// TIA Portal V17 export
// export: Created 2024-10-17T14:16:18.5693745Z, ExportSetting WithDefaults, DisplayName Totally Integrated Automation Portal, DisplayVersion V17 Update 4, DisplayName TIA Portal Openness, DisplayVersion V17 Update 4, DisplayName TIA Portal Version Control Interface, DisplayVersion V17, DisplayName SINAMICS Startdrive Advanced, DisplayVersion V17 Update2, DisplayName SINAMICS Startdrive G130, G150, S120, S150, SINAMICS MV, S210, DisplayVersion V17 Update2, DisplayName SINAMICS Startdrive G110M, G120, G120C, G120D, G120P, G115D, DisplayVersion V17 Update2, DisplayName STEP 7 Professional, DisplayVersion V17 Update 4, DisplayName STEP 7 Safety, DisplayVersion V17, DisplayName WinCC Advanced / Unified PC, DisplayVersion V17 Update 4
TYPE "LPMLV2022_typeStatusProcessVariables"
TITLE = LPMLV2022_typeStatusProcessVariables
// Support: tech.team.motioncontrol@siemens.com
// stored: IsFailsafeCompliant false
   STRUCT
      Parameter_REAL { ExternalWritable := 'False'} : Array[0.."LPMLV2022_STATUS_PROCESS_VARIABLES_PARAMETER_REAL_UPPER_LIM"] of "LPMLV2022_typeParameter_REAL";   // Structured Array of Recipe Process Variable information for values with REAL data type
      Parameter_STRING { ExternalWritable := 'False'} : Array[0.."LPMLV2022_STATUS_PROCESS_VARIABLES_PARAMETER_STRING_UPPER_LIM"] of "LPMLV2022_typeParameter_STRING";   // Structured Array of Recipe Process Variable information for values with STRING data type
      Parameter_LREAL { ExternalWritable := 'False'} : Array[0.."LPMLV2022_STATUS_PROCESS_VARIABLES_PARAMETER_LREAL_UPPER_LIM"] of "LPMLV2022_typeParameter_LREAL";   // Structured Array of Recipe Process Variable information for values with LREAL data type
      Parameter_DINT { ExternalWritable := 'False'} : Array[0.."LPMLV2022_STATUS_PROCESS_VARIABLES_PARAMETER_DINT_UPPER_LIM"] of "LPMLV2022_typeParameter_DINT";   // Structured Array of Recipe Process Variable Information for values with DINT data type
      Parameter_BOOL { ExternalWritable := 'False'} : Array[0.."LPMLV2022_STATUS_PROCESS_VARIABLES_PARAMETER_BOOL_UPPER_LIM"] of "LPMLV2022_typeParameter_BOOL";   // Structured Array of Recipe Process Variable Information for values with BOOL data type
   END_STRUCT;
END_TYPE
